FUNCTION_BLOCK AnlagenSequenz_06_ADAPTER (* Composite wrapper around AnlagenSequenz_06: DO_Mx/STOERUNG_Mx (Event+BOOL) bundled into AX adapters, ZE*_EIN/AUS each fed via its own ATM adapter socket. timeOut stays internal, not exposed. *)
  (* Standard: 61499-2; ApplicationDomain: Fördertechnik; Description: Copyright (c) 2026 HR Agrartechnik GmbH This program and the accompanying materials are made available under the terms of the Eclipse Public License 2.0 which is available at https://www.eclipse.org/legal/epl-2.0/ SPDX-License-Identifier: EPL-2.0 *)
  (* Version 1.0, 2026-08-14, Franz Höpfinger, HR Agrartechnik GmbH, initial API and implementation *)
  PACKAGE logiBUS::utils::sequence::timed;
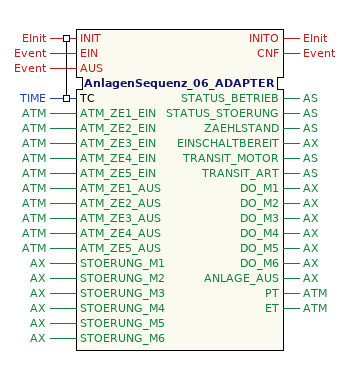
  EVENT_INPUT
    INIT : EInit WITH TC; (* Initialization Request *)
    EIN; (* Startsequenz auslösen; nur wirksam wenn EINSCHALTBEREIT=TRUE; quittiert dabei zugleich eine anstehende Störungsanzeige *)
    AUS; (* Stopsequenz auslösen, aus jedem Schritt der Vorlauf-Kette oder aus S_LAEUFT *)
  END_EVENT
  EVENT_OUTPUT
    INITO : EInit; (* Initialization Confirm *)
    CNF; (* Ausführungsbestätigung, mit jedem Zustands-Update (Werte selbst laufen ueber STATUS_BETRIEB/STATUS_STOERUNG/ZAEHLSTAND/EINSCHALTBEREIT/TRANSIT_MOTOR/TRANSIT_ART Plugs) *)
  END_EVENT
  VAR_INPUT
    TC : TIME := T#200ms; (* Cycle time for the internal TimeTicker (PT/ET readback) *)
  END_VAR
  SOCKETS
    ATM_ZE1_EIN : adapter::types::unidirectional::ATM; (* S_VOR1 zu S_VOR2, M5 startet (Vorlauf) *)
    ATM_ZE2_EIN : adapter::types::unidirectional::ATM; (* S_VOR2 zu S_VOR3, M4 startet (Vorlauf) *)
    ATM_ZE3_EIN : adapter::types::unidirectional::ATM; (* S_VOR3 zu S_VOR4, M3 startet (Vorlauf) *)
    ATM_ZE4_EIN : adapter::types::unidirectional::ATM; (* S_VOR4 zu S_VOR5, M2 startet (Vorlauf) *)
    ATM_ZE5_EIN : adapter::types::unidirectional::ATM; (* S_VOR5 zu S_LAEUFT, M1 startet (Vorlauf) *)
    ATM_ZE1_AUS : adapter::types::unidirectional::ATM; (* S_NACH1 zu S_NACH2, M2 stoppt (Nachlauf) *)
    ATM_ZE2_AUS : adapter::types::unidirectional::ATM; (* S_NACH2 zu S_NACH3, M3 stoppt (Nachlauf) *)
    ATM_ZE3_AUS : adapter::types::unidirectional::ATM; (* S_NACH3 zu S_NACH4, M4 stoppt (Nachlauf) *)
    ATM_ZE4_AUS : adapter::types::unidirectional::ATM; (* S_NACH4 zu S_NACH5, M5 stoppt (Nachlauf) *)
    ATM_ZE5_AUS : adapter::types::unidirectional::ATM; (* S_NACH5 zu S_AUS, M6 stoppt (Nachlauf) *)
    STOERUNG_M1 : adapter::types::unidirectional::AX; (* Motor 1 hat aktuell eine Störung anstehen *)
    STOERUNG_M2 : adapter::types::unidirectional::AX; (* Motor 2 hat aktuell eine Störung anstehen *)
    STOERUNG_M3 : adapter::types::unidirectional::AX; (* Motor 3 hat aktuell eine Störung anstehen *)
    STOERUNG_M4 : adapter::types::unidirectional::AX; (* Motor 4 hat aktuell eine Störung anstehen *)
    STOERUNG_M5 : adapter::types::unidirectional::AX; (* Motor 5 hat aktuell eine Störung anstehen *)
    STOERUNG_M6 : adapter::types::unidirectional::AX; (* Motor 6 hat aktuell eine Störung anstehen *)
  END_SOCKETS
  PLUGS
    STATUS_BETRIEB : adapter::types::unidirectional::AS; (* 0=Aus 1=Hochfahren 2=Läuft 3=Herunterfahren *)
    STATUS_STOERUNG : adapter::types::unidirectional::AS; (* 0=keine 4=aktiv, verriegelt bis EIN *)
    ZAEHLSTAND : adapter::types::unidirectional::AS; (* 0..6, Anzahl aktuell laufender Motoren *)
    EINSCHALTBEREIT : adapter::types::unidirectional::AX; (* TRUE nur wenn alle Motoren stehen UND alle Motoren störungsfrei sind *)
    TRANSIT_MOTOR : adapter::types::unidirectional::AS; (* 0 = keiner (S_AUS/S_LAEUFT), 1..6 = Motor-Nr., der nach Ablauf der aktuellen Zeit startet/stoppt (siehe TRANSIT_ART) *)
    TRANSIT_ART : adapter::types::unidirectional::AS; (* anlagenSequenz::TRANSIT_ART_KEINE/_VORLAUF/_NACHLAUF *)
    DO_M1 : adapter::types::unidirectional::AX; (* Laufbefehl Motor 1 *)
    DO_M2 : adapter::types::unidirectional::AX; (* Laufbefehl Motor 2 *)
    DO_M3 : adapter::types::unidirectional::AX; (* Laufbefehl Motor 3 *)
    DO_M4 : adapter::types::unidirectional::AX; (* Laufbefehl Motor 4 *)
    DO_M5 : adapter::types::unidirectional::AX; (* Laufbefehl Motor 5 *)
    DO_M6 : adapter::types::unidirectional::AX; (* Laufbefehl Motor 6 *)
    ANLAGE_AUS : adapter::types::unidirectional::AX; (* TRUE nur in S_AUS - Voraussetzung fuer Handbetrieb *)
    PT : adapter::types::unidirectional::ATM; (* Process time *)
    ET : adapter::types::unidirectional::ATM; (* Elapsed time *)
  END_PLUGS
  FBS
    Sequence : logiBUS::utils::sequence::timed::AnlagenSequenz_06;
    E_TimeOut : adapter::events::TimeOut::E_FB_TimeOut;
    TimeTicker : adapter::events::TimeOut::TimeTicker;
  END_FBS
  EVENT_CONNECTIONS
    EIN TO Sequence.EIN;
    AUS TO Sequence.AUS;
    ATM_ZE1_EIN.E1 TO Sequence.SET_ZE1_EIN;
    ATM_ZE2_EIN.E1 TO Sequence.SET_ZE2_EIN;
    ATM_ZE3_EIN.E1 TO Sequence.SET_ZE3_EIN;
    ATM_ZE4_EIN.E1 TO Sequence.SET_ZE4_EIN;
    ATM_ZE5_EIN.E1 TO Sequence.SET_ZE5_EIN;
    ATM_ZE1_AUS.E1 TO Sequence.SET_ZE1_AUS;
    ATM_ZE2_AUS.E1 TO Sequence.SET_ZE2_AUS;
    ATM_ZE3_AUS.E1 TO Sequence.SET_ZE3_AUS;
    ATM_ZE4_AUS.E1 TO Sequence.SET_ZE4_AUS;
    ATM_ZE5_AUS.E1 TO Sequence.SET_ZE5_AUS;
    STOERUNG_M1.E1 TO Sequence.EI_M1;
    STOERUNG_M2.E1 TO Sequence.EI_M2;
    STOERUNG_M3.E1 TO Sequence.EI_M3;
    STOERUNG_M4.E1 TO Sequence.EI_M4;
    STOERUNG_M5.E1 TO Sequence.EI_M5;
    STOERUNG_M6.E1 TO Sequence.EI_M6;
    Sequence.CNF TO CNF;
    Sequence.CNF TO ANLAGE_AUS.E1;
    Sequence.CNF TO STATUS_BETRIEB.E1;
    Sequence.CNF TO STATUS_STOERUNG.E1;
    Sequence.CNF TO ZAEHLSTAND.E1;
    Sequence.CNF TO EINSCHALTBEREIT.E1;
    Sequence.CNF TO TRANSIT_MOTOR.E1;
    Sequence.CNF TO TRANSIT_ART.E1;
    Sequence.EO_M1 TO DO_M1.E1;
    Sequence.EO_M2 TO DO_M2.E1;
    Sequence.EO_M3 TO DO_M3.E1;
    Sequence.EO_M4 TO DO_M4.E1;
    Sequence.EO_M5 TO DO_M5.E1;
    Sequence.EO_M6 TO DO_M6.E1;
    INIT TO Sequence.INIT;
    Sequence.INITO TO TimeTicker.INIT;
    TimeTicker.INITO TO INITO;
    TimeTicker.CNF TO ET.E1;
    TimeTicker.STARTO TO PT.E1;
  END_CONNECTIONS
  DATA_CONNECTIONS
    ATM_ZE1_EIN.D1 TO Sequence.ZE1_EIN;
    ATM_ZE2_EIN.D1 TO Sequence.ZE2_EIN;
    ATM_ZE3_EIN.D1 TO Sequence.ZE3_EIN;
    ATM_ZE4_EIN.D1 TO Sequence.ZE4_EIN;
    ATM_ZE5_EIN.D1 TO Sequence.ZE5_EIN;
    ATM_ZE1_AUS.D1 TO Sequence.ZE1_AUS;
    ATM_ZE2_AUS.D1 TO Sequence.ZE2_AUS;
    ATM_ZE3_AUS.D1 TO Sequence.ZE3_AUS;
    ATM_ZE4_AUS.D1 TO Sequence.ZE4_AUS;
    ATM_ZE5_AUS.D1 TO Sequence.ZE5_AUS;
    STOERUNG_M1.D1 TO Sequence.STOERUNG_M1;
    STOERUNG_M2.D1 TO Sequence.STOERUNG_M2;
    STOERUNG_M3.D1 TO Sequence.STOERUNG_M3;
    STOERUNG_M4.D1 TO Sequence.STOERUNG_M4;
    STOERUNG_M5.D1 TO Sequence.STOERUNG_M5;
    STOERUNG_M6.D1 TO Sequence.STOERUNG_M6;
    Sequence.STATUS_BETRIEB TO STATUS_BETRIEB.D1;
    Sequence.STATUS_STOERUNG TO STATUS_STOERUNG.D1;
    Sequence.ZAEHLSTAND TO ZAEHLSTAND.D1;
    Sequence.EINSCHALTBEREIT TO EINSCHALTBEREIT.D1;
    Sequence.TRANSIT_MOTOR TO TRANSIT_MOTOR.D1;
    Sequence.TRANSIT_ART TO TRANSIT_ART.D1;
    Sequence.ANLAGE_AUS TO ANLAGE_AUS.D1;
    Sequence.DO_M1 TO DO_M1.D1;
    Sequence.DO_M2 TO DO_M2.D1;
    Sequence.DO_M3 TO DO_M3.D1;
    Sequence.DO_M4 TO DO_M4.D1;
    Sequence.DO_M5 TO DO_M5.D1;
    Sequence.DO_M6 TO DO_M6.D1;
    TimeTicker.ET TO ET.D1;
    TimeTicker.PT TO PT.D1;
    TC TO TimeTicker.TC;
  END_CONNECTIONS
  ADAPTER_CONNECTIONS
    Sequence.timeOut TO E_TimeOut.TimeOutSocket;
    TimeTicker.TimeTickSocket TO E_TimeOut.TimeTickSocket;
  END_CONNECTIONS
END_FUNCTION_BLOCK
